// Mitsubishi GX Works2 project: STUDY-SAMPLE   PLC: Q06H

PROGRAM MAIN
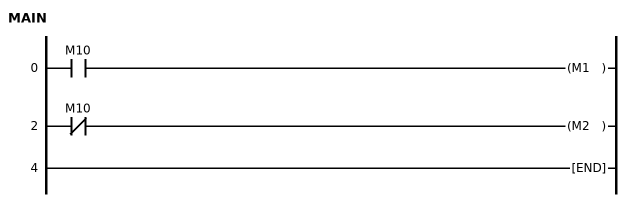
0     LD      M10
      OUT     M1
2     LDI     M10
      OUT     M2
4     END
END_PROGRAM
